(* CoDeSys 2.3.8.0 project: laserPLC.pro *)
(* Libraries: STANDARD.LIB 5.6.98 12:03:02 *)

(* Task configuration *)
TASK Standard (PRIORITY := 0, INTERVAL := T#10ms);
	MAIN
END_TASK

(* Global variable list: Globale_Variablen *)
VAR_GLOBAL

	(* schreiben *)
	TP_LaserAktiv : BOOL;
	TP_LaserHand: BOOL;
	TP_RefSetzen : BOOL;
	TP_KameraAktiv :BOOL;
	TP_MVor : BOOL;
	TP_MRueck : BOOL;
	TP_Hand: BOOL;
	TP_Auto:BOOL;
	TP_ZNullen: BOOL;
	TPKettenTyp : ARRAY[0..3] OF WORD;
	TPTypIndex: WORD;
	TPTypSpeichern: BOOL ;

	S_StUeberlast : BOOL;
	S_StLaser : BOOL;
	S_StKamera: BOOL;
	S_StKupplung:BOOL;
	S_StSpeicherSchutz:BOOL;
	S_StLaserSchutz:BOOL;
	S_StSpeicher:BOOL;
	S_StSammelStoerung:BOOL;
	S_StDruck:BOOL;
	S_StNotAus:BOOL;
	S_Frg_Sp1:BOOL;
	S_Frg_Sp2:BOOL;
	S_StRef: BOOL;

	S_MSpeicherVoll :BOOL;
	S_MSpeicherLeer:BOOL;
	S_MWarteSpeicher:BOOL;
	S_MHand :BOOL;
	S_MAuto: BOOL;
	S_MAutoStop:BOOL;

	S_FKamera:BOOL;
	S_FLaser:BOOL;

	SI_Gliederzahl : INT;
	SI_ProgNr : INT;
	SI_IO : INT;
	SI_NIO :INT;
	SI_FKamera: INT;
	SI_FLaser:INT;
	SI_FPosKamera:INT;
	SI_FPosLaser : INT;


	(* nur lesen *)
	AktTypIndex : WORD;





END_VAR

(* POU MAIN, ST *)
PROGRAM MAIN
VAR
END_VAR
;
END_PROGRAM
